// TIA Portal V19 export
FUNCTION "Input_Peripherie" : Void   // FC1010, LAD
TITLE = Input
{ S7_Optimized_Access := 'TRUE' }
// stored: AutoNumber false, SetENOAutomatically true
   VAR_TEMP
      Sperre_Inc_max : DInt;
      Sperre_Inc_min : DInt;
   END_VAR
BEGIN

REGION Network 1 (SCL): Schnelllauftor
   // Motorschutzschalter
   "Tor".In.MSS_ok := "E_MSS_ok_RT";
   // betriebsbereit
   "Tor".In.ok := "E_RT_ok";
   // Paneltasten
   "Tor".In.Knauf_Auto := "DB_ANLAGE".BA.Automat_ein;
   "Tor".In.T_auf := "Panel".RT.T_auf;
   "Tor".In.T_zu := "Panel".RT.T_zu;
   // Sensoren
   "Tor".In.S_auf := "E_S_RT_auf";
   "Tor".In.S_zu := "E_S_RT_zu";
   // --> Panel
   "Panel".RT.MSS_ok := "Tor".In.MSS_ok;
   "Panel".RT.ok := "Tor".In.ok;
   "Panel".RT.S_offen := "Tor".In.S_auf;
   "Panel".RT.S_geschlossen := "Tor".In.S_zu;
   // Automatik
   "Tor".In.Knauf_Auto := "DB_ANLAGE".BA.Automat_ein;
   // Fehlerquittung
   "Tor".In.ErrQ := "DB_ANLAGE".IN.Quitt_Err;
END_REGION

REGION Network 2 (SCL): Deckel
   REGION CM01
       // Sicherungen
       "Deckel_CM01".In.Si_24VDC_links := "E_Si_24VDC_CM01.MM01";
       "Deckel_CM01".In.Si_24VDC_rechts := "E_Si_24VDC_CM01.MM02";
       // Stellrückmeldungen
       "Deckel_CM01".In.SRM_links_auf := "E_Dkl_li_auf_CM01";
       "Deckel_CM01".In.SRM_links_zu := "E_Dkl_li_zu_CM01";
       "Deckel_CM01".In.SRM_rechts_auf := "E_Dkl_re_auf_CM01";
       "Deckel_CM01".In.SRM_rechts_zu := "E_Dkl_re_zu_CM01";
       // Sensoren
       "Deckel_CM01".In.S_links_auf := "E_S_Dkl_li_auf_CM01.BG01" AND NOT "E_S_Dkl_li_zu_CM01.BG02";
       "Deckel_CM01".In.S_links_zu := "E_S_Dkl_li_zu_CM01.BG02" AND NOT "E_S_Dkl_li_auf_CM01.BG01";
       "Deckel_CM01".In.S_rechts_auf := "E_S_Dkl_re_auf_CM01.BG03" AND NOT "E_S_Dkl_re_zu_CM01.BG04";
       "Deckel_CM01".In.S_rechts_zu := "E_S_Dkl_re_zu_CM01.BG04" AND NOT "E_S_Dkl_re_auf_CM01.BG03";
       // Bedienung via Panel
       "Deckel_CM01".In.Auto := "Panel".Deckel.CM01.Auto;
       "Deckel_CM01".In.Hand := "Panel".Deckel.CM01.Hand;
       "Deckel_CM01".In.Tipp := "Panel".Deckel.CM01.Tipp;

       "Deckel_CM01".In.T_links_auf := "Panel".Deckel.CM01.links_auf;
       "Deckel_CM01".In.T_links_zu := "Panel".Deckel.CM01.links_zu;
       "Deckel_CM01".In.T_rechts_auf := "Panel".Deckel.CM01.rechts_auf;
       "Deckel_CM01".In.T_rechts_zu := "Panel".Deckel.CM01.rechts_zu;
       // --> Panel
       "Panel".Deckel.CM01.SRM_links_auf := "Deckel_CM01".In.SRM_links_auf;
       "Panel".Deckel.CM01.SRM_links_zu := "Deckel_CM01".In.SRM_links_zu;
       "Panel".Deckel.CM01.SRM_rechts_auf := "Deckel_CM01".In.SRM_rechts_auf;
       "Panel".Deckel.CM01.SRM_rechts_zu := "Deckel_CM01".In.SRM_rechts_zu;
       "Panel".Deckel.CM01.S_links_auf := "Deckel_CM01".In.S_links_auf;
       "Panel".Deckel.CM01.S_links_zu := "Deckel_CM01".In.S_links_zu;
       "Panel".Deckel.CM01.S_rechts_auf := "Deckel_CM01".In.S_rechts_auf;
       "Panel".Deckel.CM01.S_rechts_zu := "Deckel_CM01".In.S_rechts_zu;
       "Panel".Deckel.CM01.Ist_Pos_links := "Deckel_CM01".Zst.Ist_Pos_links;
       "Panel".Deckel.CM01.Ist_Pos_rechts := "Deckel_CM01".Zst.Ist_Pos_rechts;

       // Transportwagen im sicheren Bereich
       IF "DB_Sperrbereiche".Sperre_links OR "DB_Sperrbereiche".Sperre_rechts THEN
           IF "DI_FW_1".OUT.VOR THEN
               "Deckel_CM01".Zst.TW_sicher := "DI_FW_1".ZST.PosInc >= ("DB_Sperrbereiche".Bereich[3].max_Inc + "DI_FW_1".PAR.Fahrt.Bereich_Pos);
           ELSE
               "Deckel_CM01".Zst.TW_sicher := "DI_FW_1".ZST.PosInc >= ("DB_Sperrbereiche".Bereich[3].max_Inc + "DI_FW_1".PAR.Fahrt.Bereich_lngsm);
           END_IF;
       ELSIF "DI_FW_1".OUT.VOR THEN
           "Deckel_CM01".Zst.TW_sicher := "DI_FW_1".ZST.PosInc >= ("DB_Sperrbereiche".Bereich[1].max_Inc + "DI_FW_1".PAR.Fahrt.Bereich_Pos);
       ELSE
           "Deckel_CM01".Zst.TW_sicher := "DI_FW_1".ZST.PosInc >= ("DB_Sperrbereiche".Bereich[1].max_Inc + "DI_FW_1".PAR.Fahrt.Bereich_lngsm);
       END_IF;

       // Fehlerquittung
       "Deckel_CM01".In.ErrQ := "DB_ANLAGE".IN.Quitt_Err;
   END_REGION ;
   REGION CM02
       // Sicherungen
       "Deckel_CM02".In.Si_24VDC_links := "E_Si_24VDC_CM02.MM03";
       "Deckel_CM02".In.Si_24VDC_rechts := "E_Si_24VDC_CM02.MM04";
       // Stellrückmeldungen
       "Deckel_CM02".In.SRM_links_auf := "E_Dkl_li_auf_CM02";
       "Deckel_CM02".In.SRM_links_zu := "E_Dkl_li_zu_CM02";
       "Deckel_CM02".In.SRM_rechts_auf := "E_Dkl_re_auf_CM02";
       "Deckel_CM02".In.SRM_rechts_zu := "E_Dkl_re_zu_CM02";
       // Sensoren
       "Deckel_CM02".In.S_links_auf := "E_S_Dkl_li_auf_CM02.BG12" AND NOT "E_S_Dkl_li_zu_CM02.BG13";
       "Deckel_CM02".In.S_links_zu := "E_S_Dkl_li_zu_CM02.BG13" AND NOT "E_S_Dkl_li_auf_CM02.BG12";
       "Deckel_CM02".In.S_rechts_auf := "E_S_Dkl_re_auf_CM02.BG14" AND NOT "E_S_Dkl_re_zu_CM02.BG15";
       "Deckel_CM02".In.S_rechts_zu := "E_S_Dkl_re_zu_CM02.BG15" AND NOT "E_S_Dkl_re_auf_CM02.BG14";
       // Bedienung via Panel
       "Deckel_CM02".In.Auto := "Panel".Deckel.CM02.Auto;
       "Deckel_CM02".In.Hand := "Panel".Deckel.CM02.Hand;
       "Deckel_CM02".In.Tipp := "Panel".Deckel.CM02.Tipp;

       "Deckel_CM02".In.T_links_auf := "Panel".Deckel.CM02.links_auf;
       "Deckel_CM02".In.T_links_zu := "Panel".Deckel.CM02.links_zu;
       "Deckel_CM02".In.T_rechts_auf := "Panel".Deckel.CM02.rechts_auf;
       "Deckel_CM02".In.T_rechts_zu := "Panel".Deckel.CM02.rechts_zu;
       // --> Panel
       "Panel".Deckel.CM02.SRM_links_auf := "Deckel_CM02".In.SRM_links_auf;
       "Panel".Deckel.CM02.SRM_links_zu := "Deckel_CM02".In.SRM_links_zu;
       "Panel".Deckel.CM02.SRM_rechts_auf := "Deckel_CM02".In.SRM_rechts_auf;
       "Panel".Deckel.CM02.SRM_rechts_zu := "Deckel_CM02".In.SRM_rechts_zu;
       "Panel".Deckel.CM02.S_links_auf := "Deckel_CM02".In.S_links_auf;
       "Panel".Deckel.CM02.S_links_zu := "Deckel_CM02".In.S_links_zu;
       "Panel".Deckel.CM02.S_rechts_auf := "Deckel_CM02".In.S_rechts_auf;
       "Panel".Deckel.CM02.S_rechts_zu := "Deckel_CM02".In.S_rechts_zu;
       "Panel".Deckel.CM02.Ist_Pos_links := "Deckel_CM02".Zst.Ist_Pos_links;
       "Panel".Deckel.CM02.Ist_Pos_rechts := "Deckel_CM02".Zst.Ist_Pos_rechts;

       // Transportwagen im sicheren Bereich
       IF "DB_Sperrbereiche".Sperre_links OR "DB_Sperrbereiche".Sperre_rechts THEN

           IF "DI_FW_1".OUT.VOR THEN
               "Deckel_CM02".Zst.TW_sicher :=
               ("DI_FW_1".ZST.PosInc <= ("DB_Sperrbereiche".Bereich[4].min_Inc - "DI_FW_1".PAR.Fahrt.Bereich_lngsm)) OR
               ("DI_FW_1".ZST.PosInc >= ("DB_Sperrbereiche".Bereich[4].max_Inc + "DI_FW_1".PAR.Fahrt.Bereich_Pos));

           ELSIF "DI_FW_1".OUT.RUECK THEN
               "Deckel_CM02".Zst.TW_sicher :=
               ("DI_FW_1".ZST.PosInc <= ("DB_Sperrbereiche".Bereich[4].min_Inc - "DI_FW_1".PAR.Fahrt.Bereich_Pos)) OR
               ("DI_FW_1".ZST.PosInc >= ("DB_Sperrbereiche".Bereich[4].max_Inc + "DI_FW_1".PAR.Fahrt.Bereich_lngsm));
           ELSE
               "Deckel_CM02".Zst.TW_sicher :=
               ("DI_FW_1".ZST.PosInc <= ("DB_Sperrbereiche".Bereich[4].min_Inc)) OR
               ("DI_FW_1".ZST.PosInc >= ("DB_Sperrbereiche".Bereich[4].max_Inc));
           END_IF;

       ELSIF "DI_FW_1".OUT.VOR THEN
           "Deckel_CM02".Zst.TW_sicher :=
           ("DI_FW_1".ZST.PosInc <= ("DB_Sperrbereiche".Bereich[2].min_Inc - "DI_FW_1".PAR.Fahrt.Bereich_lngsm)) OR
           ("DI_FW_1".ZST.PosInc >= ("DB_Sperrbereiche".Bereich[2].max_Inc + "DI_FW_1".PAR.Fahrt.Bereich_Pos));

       ELSIF "DI_FW_1".OUT.RUECK THEN
           "Deckel_CM02".Zst.TW_sicher :=
           ("DI_FW_1".ZST.PosInc <= ("DB_Sperrbereiche".Bereich[2].min_Inc - "DI_FW_1".PAR.Fahrt.Bereich_Pos)) OR
           ("DI_FW_1".ZST.PosInc >= ("DB_Sperrbereiche".Bereich[2].max_Inc + "DI_FW_1".PAR.Fahrt.Bereich_lngsm));

       ELSE
           "Deckel_CM02".Zst.TW_sicher :=
           ("DI_FW_1".ZST.PosInc <= ("DB_Sperrbereiche".Bereich[2].min_Inc)) OR
           ("DI_FW_1".ZST.PosInc >= ("DB_Sperrbereiche".Bereich[2].max_Inc));
       END_IF;

       // Fehlerquittung
       "Deckel_CM02".In.ErrQ := "DB_ANLAGE".IN.Quitt_Err;
   END_REGION ;
END_REGION

REGION Network 3 (SCL): CM01
   REGION Filtern
       "FP_CM01.GP01".Param.Name_Pumpe := 'FP_CM01.GP01';
       "FP_CM01.GP01".Param.Name_Filter := 'Filter HQ1';
       // Niveaus
       "FP_CM01.GP01".In.Niv_TLS := "E_Niv_TLS_CM01.BL04";
       "FP_CM01.GP01".In.Niv_min := "E_Niv_Min_CM01.BL03";
       "FP_CM01.GP01".In.Niv_max := "E_Niv_Max_CM01.BL02";
       "FP_CM01.GP01".In.Niv_Uel := NOT "E_Niv_UeL_CM01.BL01";
       "FP_CM01.GP01".In.Frg_Niv_CM05 := NOT "Pu_CM05.GP11_DB".In."Niv_max_CM05.BL01" AND NOT "Pu_CM05.GP11_DB".In."Niv_Uel_CM05.BL05";
       "FP_CM01.GP01".In.Leckage_ok := "E_LS_HQ0x.BL12";
       "FP_CM01.GP01".In.ext_Freigabe := "E_Al_Gas_ok" AND NOT "E_Not-Strom";
       // Ist-Druck Pumpe
       "FP_CM01.GP01".In.Druck_Pumpe := "Panel".IW."p_CM01.BP03";
       // Differenz-Druck Filter
       "FP_CM01.GP01".In.Delta_p_Filter := "Panel".IW."p_HQ01.BP01";

       //Stellrückmeldungen (Filtern)
       "FP_CM01.GP01".In.SRM_Saugseite_auf := "E_SRM_CM01.QM18_auf" AND NOT "E_SRM_CM01.QM18_zu";
       "FP_CM01.GP01".In.SRM_Saugseite_zu := "E_SRM_CM01.QM18_zu" AND NOT "E_SRM_CM01.QM18_auf";
       "FP_CM01.GP01".In.SRM_Eingang_Filter_auf := "E_SRM_HQ01.QM21_auf" AND NOT "E_SRM_HQ01.QM21_zu";
       "FP_CM01.GP01".In.SRM_Eingang_Filter_zu := "E_SRM_HQ01.QM21_zu" AND NOT "E_SRM_HQ01.QM21_auf";
       "FP_CM01.GP01".In.SRM_Ausgang_Filter_auf := "E_SRM_HQ01.QM23_auf" AND NOT "E_SRM_HQ01.QM23_zu";
       "FP_CM01.GP01".In.SRM_Ausgang_Filter_zu := "E_SRM_HQ01.QM23_zu" AND NOT "E_SRM_HQ01.QM23_auf";

       "FP_CM01.GP01".In.SRM_Eingang_Spülltg_P_auf := "E_SRM_CM01.QM19_auf" AND NOT "E_SRM_CM01.QM19_zu";
       "FP_CM01.GP01".In.SRM_Eingang_Spülltg_P_zu := "E_SRM_CM01.QM19_zu" AND NOT "E_SRM_CM01.QM19_auf";
       "FP_CM01.GP01".In.SRM_Eingang_Spülltg_F_auf := "E_SRM_HQ01.QM22_auf" AND NOT "E_SRM_HQ01.QM22_zu";
       "FP_CM01.GP01".In.SRM_Eingang_Spülltg_F_zu := "E_SRM_HQ01.QM22_zu" AND NOT "E_SRM_HQ01.QM22_auf";
       "FP_CM01.GP01".In.SRM_Ausgang_Spülltg_auf := "E_SRM_HQ01.QM24_auf" AND NOT "E_SRM_HQ01.QM24_zu";
       "FP_CM01.GP01".In.SRM_Ausgang_Spülltg_zu := "E_SRM_HQ01.QM24_zu" AND NOT "E_SRM_HQ01.QM24_auf";
       "FP_CM01.GP01".In.SRM_Entluften_auf := "E_SRM_HQ01.LV01_auf" AND NOT "E_SRM_HQ01.LV01_zu";
       "FP_CM01.GP01".In.SRM_Entlueften_zu := "E_SRM_HQ01.LV01_zu" AND NOT "E_SRM_HQ01.LV01_auf";

       // Filtergehäuse
       "FP_CM01.GP01".In.GW_p_FG := "E_GW_p_HQ01.BP01";
       "FP_CM01.GP01".In.Sensor_FG_links := "E_S_FG_li_HQ01.BG07";
       "FP_CM01.GP01".In.Sensor_FG_rechts := "E_S_FG_re_HQ01.BG08";
       "FP_CM01.GP01".In.Einhausung_HQ0x_zu := "DB_PNOZ_IN_Out".In.FG_zu_HQ01;
       "FP_CM01.GP01".Param.WarnGr_FW := "Panel".HQ01.WarnGr_FW;
       "FP_CM01.GP01".Param.Wechsel_FW := "Panel".HQ01.Wechsel_FW;

       // Not-Halt
       "FP_CM01.GP01".In.NotHalt := NOT "DB_PNOZ_IN_Out".In.NH_Frg_FP_CM01;

       "FP_CM01.GP01".In.GW_p_FP := "E_GW_p_CM01.BP03";
       "FP_CM01.GP01".In.GW_LF_FP := "E_GW_LF_CM01.BN01";

       // Frequenzumrichter [Index 1] 
       "FP_CM01.GP01".In.FU_speed := "FU_In_Out".FU[1].PE.Speed;
       "FP_CM01.GP01".In.FU_betriebsbereit := "FU_In_Out".FU[1].PE.Statusbyte.Bereit;
       "FP_CM01.GP01".In.FU_Stoerung := "FU_In_Out".FU[1].PE.Statusbyte.Stoer;
       "FP_CM01.GP01".Param.SW_Hand := "Panel".FP_CM01.SW_Hand;
       "FP_CM01.GP01".Param.SW_Auto_AZ := "Panel".FP_CM01.SW_Auto_AZ;
       "FP_CM01.GP01".Param.SW_Auto_aAZ := "Panel".FP_CM01.SW_Auto_aAZ;

       // Hand
       "FP_CM01.GP01".In.Ein := "Panel".FP_CM01.Ein;
       // Auto
       "FP_CM01.GP01".In.Auto := "Panel".FP_CM01.Auto;
       // Betriebsart
       "FP_CM01.GP01".In.Betriebsart := "Panel".FP_CM01.BA;
       // Spülzeit
       "FP_CM01.GP01".Param.Spülzeit_Pumpe := DINT_TO_TIME(INT_TO_DINT("Panel".FP_CM01.Sp_Ventil.Sollzeit) * 1000);
       // Zeiten Filterwechsel
       "FP_CM01.GP01".Param.FG_Zeit_leeren_Saurebecken := DINT_TO_TIME(INT_TO_DINT("Panel".FP_CM01.Sp_Filter.Zeit_leeren_Saure) * 1000);
       "FP_CM01.GP01".Param.FG_Zeit_leeren_CM05 := DINT_TO_TIME(INT_TO_DINT("Panel".FP_CM01.Sp_Filter.Zeit_leeren_CM05) * 1000);
       "FP_CM01.GP01".Param.FW_Spülzeit := DINT_TO_TIME(INT_TO_DINT("Panel".FP_CM01.Sp_Filter.Zeit_Spülen) * 1000);
       "FP_CM01.GP01".Param.FW_Wartezeit := DINT_TO_TIME(INT_TO_DINT("Panel".FP_CM01.Sp_Filter.Wartezeit) * 1000);
       "FP_CM01.GP01".Param.FW_Zeit_fuellen := DINT_TO_TIME(INT_TO_DINT("Panel".FP_CM01.Sp_Filter.Zeit_füllen) * 1000);
       // Drucktest Pumpe
       "FP_CM01.GP01".Param.DT_Druckaufbau := T#1m;
       "FP_CM01.GP01".Param.SW_Drucktest_Pumpe := "Panel".FP_CM01.Drucktest_Pumpe.Solldruck;
       "FP_CM01.GP01".Param.DT_Testzeit_Pumpe := DINT_TO_TIME(INT_TO_DINT("Panel".FP_CM01.Drucktest_Pumpe.Sollzeit) * 1000);
       // Drucktest Filter
       "FP_CM01.GP01".Param.DT_Druckaufbau := T#1m;
       "FP_CM01.GP01".Param.SW_Drucktest_Filter := "Panel".FP_CM01.Drucktest_Filter.Solldruck;
       "FP_CM01.GP01".Param.DT_Testzeit_Filter := DINT_TO_TIME(INT_TO_DINT("Panel".FP_CM01.Drucktest_Filter.Sollzeit) * 1000);

       IF "Panel".HQ01.Quitt_FW THEN
           "FP_CM01.GP01".In.Quitt_FW := TRUE;
           "Panel".HQ01.Quitt_FW := FALSE;
       END_IF;

       //--> Panel
       "Panel".CM01.GW_p_FP := "FP_CM01.GP01".Mld.GW_p_FP;
       "Panel".CM01.GW_LF_FP := "FP_CM01.GP01".Mld.GW_LF_FP;

       "Panel".FP_CM01.Sp_Ventil.Restzeit := TIME_TO_INT("FP_CM01.GP01".Zst.Restzeit_Spülen_Pumpe / 1000);
       "Panel".FP_CM01.Sp_Filter.Restzeit := TIME_TO_INT("FP_CM01.GP01".Zst.Restzeit_Filter / 1000);
       "Panel".FP_CM01.Drucktest_Pumpe.Restzeit := TIME_TO_INT("FP_CM01.GP01".Zst.Restzeit_DT / 1000);
       "Panel".FP_CM01.Drucktest_Pumpe.Schritt := "FP_CM01.GP01".Zst.Status_DT_Pumpe;
       "Panel".FP_CM01.Status_FW := "FP_CM01.GP01".Zst.Status_FW;

       "Panel".FP_CM01.Bedienung_Erlaubt := "FP_CM01.GP01".Zst.Bedienung_erlaubt;

       "Panel".FP_CM01.Status := "FP_CM01.GP01".Zst.Status_GP0x;
       "Panel".FP_CM01.speed := "FP_CM01.GP01".Zst.speed;

       "Panel".HQ01.S_Dkl_FG_li := "FP_CM01.GP01".In.Sensor_FG_links;
       "Panel".HQ01.S_Dkl_FG_re := "FP_CM01.GP01".In.Sensor_FG_rechts;
       "Panel".HQ01.S_FG_zu := "FP_CM01.GP01".In.Einhausung_HQ0x_zu;
       "Panel".HQ01.Niv_Leckage := NOT "FP_CM01.GP01".In.Leckage_ok;
       "Panel".HQ01.Quitt_FW_erlaubt := "FP_CM01.GP01".In.Sensor_FG_links AND "FP_CM01.GP01".In.Sensor_FG_rechts AND
       "FP_CM01.GP01".In.Einhausung_HQ0x_zu AND "FP_CM01.GP01".Mld.FG_Spülen_Ende AND "FP_CM01.GP01".Zst.Status_FW = 5;

       "Panel".FP_CM01.Drucktest_Filter.Restzeit := TIME_TO_INT("FP_CM01.GP01".Zst.Restzeit_DT / 1000);
       "Panel".FP_CM01.Drucktest_Filter.Schritt := "FP_CM01.GP01".Zst.Status_DT_Filter;
   END_REGION

   REGION Umwälzen
       "UP_CM01.GP02".Param.Name := 'UP_CM01.GP02';
       // Niveaus
       "UP_CM01.GP02".In.Niv_TLS := "E_Niv_TLS_CM01.BL04";
       "UP_CM01.GP02".In.Niv_min := "E_Niv_Min_CM01.BL03";
       "UP_CM01.GP02".In.Niv_max := "E_Niv_Max_CM01.BL02";
       "UP_CM01.GP02".In.Niv_Uel := NOT "E_Niv_UeL_CM01.BL01";
       "UP_CM01.GP02".In.Frg_Niv_CM05 := NOT "Pu_CM05.GP11_DB".In."Niv_max_CM05.BL01" AND NOT "Pu_CM05.GP11_DB".In."Niv_Uel_CM05.BL05";
       "UP_CM01.GP02".In.ext_Freigabe := "E_Al_Gas_ok" AND NOT "E_Not-Strom";
       // Ist-Druck
       "UP_CM01.GP02".In.Druck_Pumpe := "Panel".IW."p_CM01.BP04";

       //Stellrückmeldungen (Umwälzen)
       "UP_CM01.GP02".In.SRM_Saugseite_auf := "E_SRM_CM01.QM25_auf" AND NOT "E_SRM_CM01.QM25_zu";
       "UP_CM01.GP02".In.SRM_Saugseite_zu := "E_SRM_CM01.QM25_zu" AND NOT "E_SRM_CM01.QM25_auf";
       "UP_CM01.GP02".In.SRM_Druckseite_auf := "E_SRM_CM01.QM26_auf" AND NOT "E_SRM_CM01.QM26_zu";
       "UP_CM01.GP02".In.SRM_Druckseite_zu := "E_SRM_CM01.QM26_zu" AND NOT "E_SRM_CM01.QM26_auf";
       "UP_CM01.GP02".In.SRM_Eingang_Spülltg_auf := "E_SRM_CM01.QM20_auf" AND NOT "E_SRM_CM01.QM20_zu";
       "UP_CM01.GP02".In.SRM_Eingang_Spülltg_zu := "E_SRM_CM01.QM20_zu" AND NOT "E_SRM_CM01.QM20_auf";
       "UP_CM01.GP02".In.SRM_Ausgang_Spülltg_auf := "E_SRM_CM01.QM27_auf" AND NOT "E_SRM_CM01.QM27_zu";
       "UP_CM01.GP02".In.SRM_Ausgang_Spülltg_zu := "E_SRM_CM01.QM27_zu" AND NOT "E_SRM_CM01.QM27_auf";
       "UP_CM01.GP02".In.SRM_Entsogung_UV02_auf := "E_SRM_GP02.QM45_auf" AND NOT "E_SRM_GP02.QM45_zu";
       "UP_CM01.GP02".In.SRM_Entsogung_UV02_zu := "E_SRM_GP02.QM45_zu" AND NOT "E_SRM_GP02.QM45_auf";
       "UP_CM01.GP02".In.SRM_UV02_GP01_auf := "DB_PNOZ_IN_Out".In."SRM_Auf_BG-QM44" AND NOT "DB_PNOZ_IN_Out".In."SRM_Zu_BG-QM44";
       "UP_CM01.GP02".In.SRM_UV02_GP01_zu := "DB_PNOZ_IN_Out".In."SRM_Zu_BG-QM44" AND NOT "DB_PNOZ_IN_Out".In."SRM_Auf_BG-QM44";
       "UP_CM01.GP02".In.SRM_UV02_GP02_auf := "DB_PNOZ_IN_Out".In."SRM_Auf_BG-QM43" AND NOT "DB_PNOZ_IN_Out".In."SRM_Zu_BG-QM43";
       "UP_CM01.GP02".In.SRM_UV02_GP02_zu := "DB_PNOZ_IN_Out".In."SRM_Zu_BG-QM43" AND NOT "DB_PNOZ_IN_Out".In."SRM_Auf_BG-QM43";
       "UP_CM01.GP02".In."SRM_GP02.QM41_auf" := "E_SRM_GP02.QM41_auf" AND NOT "E_SRM_GP02.QM41_zu";
       "UP_CM01.GP02".In."SRM_GP01.QM14_auf" := "E_SRM_GP01.QM14_auf" AND NOT "E_SRM_GP01.QM14_zu";

       // Türen GP0x
       "UP_CM01.GP02".In.Tuer_zu_Seite_GP01 := "DB_PNOZ_IN_Out".In.Tuer_zu_Seite_GP01;
       "UP_CM01.GP02".In.Tuer_zu_vorn_GP01 := "DB_PNOZ_IN_Out".In.Tuer_zu_vorn_GP01;
       "UP_CM01.GP02".In.Tuer_zu_vorn_GP02 := "DB_PNOZ_IN_Out".In.Tuer_zu_vorn_GP02;
       // Leckagen Entsorgung
       "UP_CM01.GP02".In.Leckage_Doppelrohr_ok_BL26 := "E_LS_GP02.BL26";
       "UP_CM01.GP02".In.Leckage_Doppelschlauch_ok_BL33 := "E_LS_GP02.BL33";
       "UP_CM01.GP02".In.Leckage_Uml_Tunnel_ok_BL34 := "E_LS_GP01.BL34";
       "UP_CM01.GP02".In.Leckage_PFA_Uebergang_ok_BL16 := "E_LS_GP01.BL16";
       "UP_CM01.GP02".In.Leckage_PFA_Uebergang_ok_BL25 := "E_LS_GP02.BL25";

       "UP_CM01.GP02".In.Imp_Dfl := "E_Imp_GP02.BF02";
       "UP_CM01.GP02".In.Quitt_Al_Dfl := "DB_ANLAGE".IN.Quitt_Err;

       "UP_CM01.GP02".In.GW_p_UP := "E_GW_p_CM01.BP04";
       "UP_CM01.GP02".In.GW_LF_UP := "E_GW_LF_CM01.BN02";
       "UP_CM01.GP02".In.GW_Dfl := "E_GW_Dfl_GP02.BF02";
       // TW senkt
       "UP_CM01.GP02".In.TW_senkt := ("DB_POS".POS[1].FW_Senkt OR "DB_POS".POS[2].FW_Senkt OR "DB_POS".POS[3].FW_Senkt
       OR "DB_POS".POS[4].FW_Senkt OR "DB_POS".POS[5].FW_Senkt OR "DB_POS".POS[6].FW_Senkt) AND "DI_FW_1".ZST.Mittig;

       // Frequenzumrichter [Index 2] Umwälzen
       "UP_CM01.GP02".In.FU_speed := "FU_In_Out".FU[2].PE.Speed;
       "UP_CM01.GP02".In.FU_betriebsbereit := "FU_In_Out".FU[2].PE.Statusbyte.Bereit;
       "UP_CM01.GP02".In.FU_Stoerung := "FU_In_Out".FU[2].PE.Statusbyte.Stoer;
       "UP_CM01.GP02".Param.SW_Hand := "Panel".UP_CM01.SW_Hand;
       "UP_CM01.GP02".Param.SW_Auto_AZ := "Panel".UP_CM01.SW_Auto_AZ;
       "UP_CM01.GP02".Param.SW_Auto_aAZ := "Panel".UP_CM01.SW_Auto_aAZ;

       // Hand
       "UP_CM01.GP02".In.Ein := "Panel".UP_CM01.Ein;
       // Auto
       "UP_CM01.GP02".In.Auto := "Panel".UP_CM01.Auto;
       // Betriebsart
       "UP_CM01.GP02".In.Betriebsart := "Panel".UP_CM01.BA;
       // Spülzeit
       "UP_CM01.GP02".Param.Spülzeit := DINT_TO_TIME(INT_TO_DINT("Panel".UP_CM01.Sp_Ventil.Sollzeit) * 1000);
       // Drucktest
       "UP_CM01.GP02".Param.DT_Druckaufbau := T#1m;
       "UP_CM01.GP02".Param.SW_Drucktest := "Panel".UP_CM01.Drucktest.Solldruck;
       "UP_CM01.GP02".Param.DT_Testzeit := DINT_TO_TIME(INT_TO_DINT("Panel".UP_CM01.Drucktest.Sollzeit) * 1000);

       //--> Panel
       "Panel".CM01.Niv_TGS := "UP_CM01.GP02".In.Niv_TLS;
       "Panel".CM01.Niv_Min := "UP_CM01.GP02".In.Niv_min;
       "Panel".CM01.Niv_max := "UP_CM01.GP02".In.Niv_max;
       "Panel".CM01.Niv_Uel := "UP_CM01.GP02".Mld.Niv_Ueberlauf;
       "Panel".CM01.GW_p_UP := "UP_CM01.GP02".Mld.GW_p_UP;
       "Panel".CM01.GW_LF_UP := "UP_CM01.GP02".Mld.GW_LF_UP;
       "Panel".CM01.Niv_Proz := "UP_CM01.GP02".Zst.Niveau;
       "Panel".UP_CM01.Sp_Ventil.Restzeit := TIME_TO_INT("UP_CM01.GP02".Zst.Restzeit_Spülen / 1000);
       "Panel".UP_CM01.Drucktest.Restzeit := TIME_TO_INT("UP_CM01.GP02".Zst.Restzeit_DT / 1000);
       "Panel".UP_CM01.Drucktest.Schritt := "UP_CM01.GP02".Zst.Status_DT;
       "Panel".UP_CM01.Status := "UP_CM01.GP02".Zst.Status_GP0x;
       "Panel".UP_CM01.speed := "UP_CM01.GP02".Zst.speed;
       "Panel".UP_CM01.Bedienung_Erlaubt := "UP_CM01.GP02".Zst.Bedienung_erlaubt;
   END_REGION
END_REGION

REGION Network 4 (SCL): CM02
   REGION Filtern
       "FP_CM02.GP04".Param.Name_Pumpe := 'FP_CM02.GP04';
       "FP_CM02.GP04".Param.Name_Filter := 'Filter HQ2';
       // Niveaus
       "FP_CM02.GP04".In.Niv_TLS := "E_Niv_TLS_CM02.BL11";
       "FP_CM02.GP04".In.Niv_min := "E_Niv_Min_CM02.BL10";
       "FP_CM02.GP04".In.Niv_max := "E_Niv_Max_CM02.BL09";
       "FP_CM02.GP04".In.Niv_Uel := NOT "E_Niv_UeL_CM02.BL08";
       "FP_CM02.GP04".In.Frg_Niv_CM05 := NOT "Pu_CM05.GP11_DB".In."Niv_max_CM05.BL01" AND NOT "Pu_CM05.GP11_DB".In."Niv_Uel_CM05.BL05";
       "FP_CM02.GP04".In.Leckage_ok := "E_LS_HQ0x.BL12";
       "FP_CM02.GP04".In.ext_Freigabe := "E_Al_Gas_ok" AND NOT "E_Not-Strom";
       // Ist-Druck Pumpe
       "FP_CM02.GP04".In.Druck_Pumpe := "Panel".IW."p_CM02.BP06";
       // Differenz-Druck Filter
       "FP_CM02.GP04".In.Delta_p_Filter := "Panel".IW."p_HQ02.BP02";

       //Stellrückmeldungen (Filtern)
       "FP_CM02.GP04".In.SRM_Saugseite_auf := "E_SRM_CM02.QM55_auf" AND NOT "E_SRM_CM02.QM55_zu";
       "FP_CM02.GP04".In.SRM_Saugseite_zu := "E_SRM_CM02.QM55_zu" AND NOT "E_SRM_CM02.QM55_auf";
       "FP_CM02.GP04".In.SRM_Eingang_Filter_auf := "E_SRM_HQ02.QM59_auf" AND NOT "E_SRM_HQ02.QM59_zu";
       "FP_CM02.GP04".In.SRM_Eingang_Filter_zu := "E_SRM_HQ02.QM59_zu" AND NOT "E_SRM_HQ02.QM59_auf";
       "FP_CM02.GP04".In.SRM_Ausgang_Filter_auf := "E_SRM_HQ02.QM60_auf" AND NOT "E_SRM_HQ02.QM60_zu";
       "FP_CM02.GP04".In.SRM_Ausgang_Filter_zu := "E_SRM_HQ02.QM60_zu" AND NOT "E_SRM_HQ02.QM60_auf";

       "FP_CM02.GP04".In.SRM_Eingang_Spülltg_P_auf := "E_SRM_CM02.QM56_auf" AND NOT "E_SRM_CM02.QM56_zu";
       "FP_CM02.GP04".In.SRM_Eingang_Spülltg_P_zu := "E_SRM_CM02.QM56_zu" AND NOT "E_SRM_CM02.QM56_auf";
       "FP_CM02.GP04".In.SRM_Eingang_Spülltg_F_auf := "E_SRM_HQ02.QM58_auf" AND NOT "E_SRM_HQ02.QM58_zu";
       "FP_CM02.GP04".In.SRM_Eingang_Spülltg_F_zu := "E_SRM_HQ02.QM58_zu" AND NOT "E_SRM_HQ02.QM58_auf";
       "FP_CM02.GP04".In.SRM_Ausgang_Spülltg_auf := "E_SRM_HQ02.QM61_auf" AND NOT "E_SRM_HQ02.QM61_zu";
       "FP_CM02.GP04".In.SRM_Ausgang_Spülltg_zu := "E_SRM_HQ02.QM61_zu" AND NOT "E_SRM_HQ02.QM61_auf";
       "FP_CM02.GP04".In.SRM_Entluften_auf := "E_SRM_HQ02.LV02_auf" AND NOT "E_SRM_HQ02.LV02_zu";
       "FP_CM02.GP04".In.SRM_Entlueften_zu := "E_SRM_HQ02.LV02_zu" AND NOT "E_SRM_HQ02.LV02_auf";

       // Filtergehäuse
       "FP_CM02.GP04".In.GW_p_FG := "E_GW_p_HQ02.BP02";
       "FP_CM02.GP04".In.Sensor_FG_links := "E_S_FG_li_HQ02.BG10";
       "FP_CM02.GP04".In.Sensor_FG_rechts := "E_S_FG_re_HQ02.BG11";
       "FP_CM02.GP04".In.Einhausung_HQ0x_zu := "DB_PNOZ_IN_Out".In.FG_zu_HQ02;
       "FP_CM02.GP04".Param.WarnGr_FW := "Panel".HQ02.WarnGr_FW;
       "FP_CM02.GP04".Param.Wechsel_FW := "Panel".HQ02.Wechsel_FW;

       // Not-Halt
       "FP_CM02.GP04".In.NotHalt := NOT "DB_PNOZ_IN_Out".In.NH_Frg_FP_CM02;

       "FP_CM02.GP04".In.GW_p_FP := "E_GW_p_CM02.BP06";
       "FP_CM02.GP04".In.GW_LF_FP := "E_GW_LF_CM02.BN03";

       // Frequenzumrichter [Index 4] 
       "FP_CM02.GP04".In.FU_speed := "FU_In_Out".FU[4].PE.Speed;
       "FP_CM02.GP04".In.FU_betriebsbereit := "FU_In_Out".FU[4].PE.Statusbyte.Bereit;
       "FP_CM02.GP04".In.FU_Stoerung := "FU_In_Out".FU[4].PE.Statusbyte.Stoer;
       "FP_CM02.GP04".Param.SW_Hand := "Panel".FP_CM02.SW_Hand;
       "FP_CM02.GP04".Param.SW_Auto_AZ := "Panel".FP_CM02.SW_Auto_AZ;
       "FP_CM02.GP04".Param.SW_Auto_aAZ := "Panel".FP_CM02.SW_Auto_aAZ;

       // Hand
       "FP_CM02.GP04".In.Ein := "Panel".FP_CM02.Ein;
       // Auto
       "FP_CM02.GP04".In.Auto := "Panel".FP_CM02.Auto;
       // Betriebsart
       "FP_CM02.GP04".In.Betriebsart := "Panel".FP_CM02.BA;
       // Spülzeit
       "FP_CM02.GP04".Param.Spülzeit_Pumpe := DINT_TO_TIME(INT_TO_DINT("Panel".FP_CM02.Sp_Ventil.Sollzeit) * 1000);
       // Zeiten Filterwechsel
       "FP_CM02.GP04".Param.FG_Zeit_leeren_Saurebecken := DINT_TO_TIME(INT_TO_DINT("Panel".FP_CM02.Sp_Filter.Zeit_leeren_Saure) * 1000);
       "FP_CM02.GP04".Param.FG_Zeit_leeren_CM05 := DINT_TO_TIME(INT_TO_DINT("Panel".FP_CM02.Sp_Filter.Zeit_leeren_CM05) * 1000);
       "FP_CM02.GP04".Param.FW_Spülzeit := DINT_TO_TIME(INT_TO_DINT("Panel".FP_CM02.Sp_Filter.Zeit_Spülen) * 1000);
       "FP_CM02.GP04".Param.FW_Wartezeit := DINT_TO_TIME(INT_TO_DINT("Panel".FP_CM02.Sp_Filter.Wartezeit) * 1000);
       "FP_CM02.GP04".Param.FW_Zeit_fuellen := DINT_TO_TIME(INT_TO_DINT("Panel".FP_CM02.Sp_Filter.Zeit_füllen) * 1000);
       "Panel".FP_CM02.Status_FW := "FP_CM02.GP04".Zst.Status_FW;
       // Drucktest Pumpe
       "FP_CM02.GP04".Param.DT_Druckaufbau := T#1m;
       "FP_CM02.GP04".Param.SW_Drucktest_Pumpe := "Panel".FP_CM02.Drucktest_Pumpe.Solldruck;
       "FP_CM02.GP04".Param.DT_Testzeit_Pumpe := DINT_TO_TIME(INT_TO_DINT("Panel".FP_CM02.Drucktest_Pumpe.Sollzeit) * 1000);
       // Drucktest Filter
       "FP_CM02.GP04".Param.DT_Druckaufbau := T#1m;
       "FP_CM02.GP04".Param.SW_Drucktest_Filter := "Panel".FP_CM02.Drucktest_Filter.Solldruck;
       "FP_CM02.GP04".Param.DT_Testzeit_Filter := DINT_TO_TIME(INT_TO_DINT("Panel".FP_CM02.Drucktest_Filter.Sollzeit) * 1000);

       IF "Panel".HQ02.Quitt_FW THEN
           "FP_CM02.GP04".In.Quitt_FW := TRUE;
           "Panel".HQ02.Quitt_FW := FALSE;
       END_IF;

       //--> Panel
       "Panel".CM02.GW_p_FP := "FP_CM02.GP04".Mld.GW_p_FP;
       "Panel".CM02.GW_LF_FP := "FP_CM02.GP04".Mld.GW_LF_FP;

       "Panel".FP_CM02.Sp_Ventil.Restzeit := TIME_TO_INT("FP_CM02.GP04".Zst.Restzeit_Spülen_Pumpe / 1000);
       "Panel".FP_CM02.Sp_Filter.Restzeit := TIME_TO_INT("FP_CM02.GP04".Zst.Restzeit_Filter / 1000);
       "Panel".FP_CM02.Drucktest_Pumpe.Restzeit := TIME_TO_INT("FP_CM02.GP04".Zst.Restzeit_DT / 1000);
       "Panel".FP_CM02.Drucktest_Pumpe.Schritt := "FP_CM02.GP04".Zst.Status_DT_Pumpe;
       "Panel".FP_CM02.Status := "FP_CM02.GP04".Zst.Status_GP0x;
       "Panel".FP_CM02.speed := "FP_CM02.GP04".Zst.speed;

       "Panel".FP_CM02.Bedienung_Erlaubt := "FP_CM02.GP04".Zst.Bedienung_erlaubt;

       "Panel".HQ02.S_Dkl_FG_li := "FP_CM02.GP04".In.Sensor_FG_links;
       "Panel".HQ02.S_Dkl_FG_re := "FP_CM02.GP04".In.Sensor_FG_rechts;
       "Panel".HQ02.S_FG_zu := "FP_CM02.GP04".In.Einhausung_HQ0x_zu;
       "Panel".HQ02.Niv_Leckage := NOT "FP_CM02.GP04".In.Leckage_ok;

       "Panel".HQ02.Quitt_FW_erlaubt := "FP_CM02.GP04".In.Sensor_FG_links AND "FP_CM02.GP04".In.Sensor_FG_rechts AND
       "FP_CM02.GP04".In.Einhausung_HQ0x_zu AND "FP_CM02.GP04".Mld.FG_Spülen_Ende AND "FP_CM02.GP04".Zst.Status_FW = 5;

       "Panel".FP_CM02.Drucktest_Filter.Restzeit := TIME_TO_INT("FP_CM02.GP04".Zst.Restzeit_DT / 1000);
       "Panel".FP_CM02.Drucktest_Filter.Schritt := "FP_CM02.GP04".Zst.Status_DT_Filter;
   END_REGION

   REGION Umwälzen
       "UP_CM02.GP05".Param.Name := 'UP_CM02.GP05';
       // Niveaus
       "UP_CM02.GP05".In.Niv_TLS := "E_Niv_TLS_CM02.BL11";
       "UP_CM02.GP05".In.Niv_min := "E_Niv_Min_CM02.BL10";
       "UP_CM02.GP05".In.Niv_max := "E_Niv_Max_CM02.BL09";
       "UP_CM02.GP05".In.Niv_Uel := NOT "E_Niv_UeL_CM02.BL08";
       "UP_CM02.GP05".In.Frg_Niv_CM05 := NOT "Pu_CM05.GP11_DB".In."Niv_max_CM05.BL01" AND NOT "Pu_CM05.GP11_DB".In."Niv_Uel_CM05.BL05";
       "UP_CM02.GP05".In.ext_Freigabe := "E_Al_Gas_ok" AND NOT "E_Not-Strom";
       // Ist-Druck
       "UP_CM02.GP05".In.Druck_Pumpe := "Panel".IW."p_CM02.BP07";

       //Stellrückmeldungen
       "UP_CM02.GP05".In.SRM_Saugseite_auf := "E_SRM_CM02.QM62_auf" AND NOT "E_SRM_CM02.QM62_zu";
       "UP_CM02.GP05".In.SRM_Saugseite_zu := "E_SRM_CM02.QM62_zu" AND NOT "E_SRM_CM02.QM62_auf";
       "UP_CM02.GP05".In.SRM_Druckseite_auf := "E_SRM_CM02.QM63_auf" AND NOT "E_SRM_CM02.QM63_zu";
       "UP_CM02.GP05".In.SRM_Druckseite_zu := "E_SRM_CM02.QM63_zu" AND NOT "E_SRM_CM02.QM63_auf";
       "UP_CM02.GP05".In.SRM_Eingang_Spülltg_auf := "E_SRM_CM02.QM57_auf" AND NOT "E_SRM_CM02.QM57_zu";
       "UP_CM02.GP05".In.SRM_Eingang_Spülltg_zu := "E_SRM_CM02.QM57_zu" AND NOT "E_SRM_CM02.QM57_auf";
       "UP_CM02.GP05".In.SRM_Ausgang_Spülltg_auf := "E_SRM_CM02.QM64_auf" AND NOT "E_SRM_CM02.QM64_zu";
       "UP_CM02.GP05".In.SRM_Ausgang_Spülltg_zu := "E_SRM_CM02.QM64_zu" AND NOT "E_SRM_CM02.QM64_auf";
       "UP_CM02.GP05".In.SRM_Entsogung_UV02_auf := "E_SRM_GP02.QM46_auf" AND NOT "E_SRM_GP02.QM46_zu";
       "UP_CM02.GP05".In.SRM_Entsogung_UV02_zu := "E_SRM_GP02.QM46_zu" AND NOT "E_SRM_GP02.QM46_auf";
       "UP_CM02.GP05".In.SRM_UV02_GP01_auf := "DB_PNOZ_IN_Out".In."SRM_Auf_BG-QM44" AND NOT "DB_PNOZ_IN_Out".In."SRM_Zu_BG-QM44";
       "UP_CM02.GP05".In.SRM_UV02_GP01_zu := "DB_PNOZ_IN_Out".In."SRM_Zu_BG-QM44" AND NOT "DB_PNOZ_IN_Out".In."SRM_Auf_BG-QM44";
       "UP_CM02.GP05".In.SRM_UV02_GP02_auf := "DB_PNOZ_IN_Out".In."SRM_Auf_BG-QM43" AND NOT "DB_PNOZ_IN_Out".In."SRM_Zu_BG-QM43";
       "UP_CM02.GP05".In.SRM_UV02_GP02_zu := "DB_PNOZ_IN_Out".In."SRM_Zu_BG-QM43" AND NOT "DB_PNOZ_IN_Out".In."SRM_Auf_BG-QM43";
       "UP_CM02.GP05".In."SRM_GP02.QM41_auf" := "E_SRM_GP02.QM41_auf" AND NOT "E_SRM_GP02.QM41_zu";
       "UP_CM02.GP05".In."SRM_GP01.QM14_auf" := "E_SRM_GP01.QM14_auf" AND NOT "E_SRM_GP01.QM14_zu";

       // Türen GP0x
       "UP_CM02.GP05".In.Tuer_zu_Seite_GP01 := "DB_PNOZ_IN_Out".In.Tuer_zu_Seite_GP01;
       "UP_CM02.GP05".In.Tuer_zu_vorn_GP01 := "DB_PNOZ_IN_Out".In.Tuer_zu_vorn_GP01;
       "UP_CM02.GP05".In.Tuer_zu_vorn_GP02 := "DB_PNOZ_IN_Out".In.Tuer_zu_vorn_GP02;

       // Leckagen Entsorgung
       "UP_CM02.GP05".In.Leckage_Doppelrohr_ok_BL26 := "E_LS_GP02.BL26";
       "UP_CM02.GP05".In.Leckage_Doppelschlauch_ok_BL33 := "E_LS_GP02.BL33";
       "UP_CM02.GP05".In.Leckage_Uml_Tunnel_ok_BL34 := "E_LS_GP01.BL34";
       "UP_CM02.GP05".In.Leckage_PFA_Uebergang_ok_BL16 := "E_LS_GP01.BL16";
       "UP_CM02.GP05".In.Leckage_PFA_Uebergang_ok_BL25 := "E_LS_GP02.BL25";

       "UP_CM02.GP05".In.Imp_Dfl := "E_Imp_GP02.BF02";
       "UP_CM02.GP05".In.Quitt_Al_Dfl := "DB_ANLAGE".IN.Quitt_Err;

       "UP_CM02.GP05".In.GW_p_UP := "E_GW_p_CM02.BP07";
       "UP_CM02.GP05".In.GW_p_UP := "E_GW_LF_CM02.BN04";
       "UP_CM02.GP05".In.GW_Dfl := "E_GW_Dfl_GP02.BF02";
       // TW senkt
       "UP_CM02.GP05".In.TW_senkt := ("DB_POS".POS[13].FW_Senkt OR "DB_POS".POS[14].FW_Senkt OR "DB_POS".POS[15].FW_Senkt
       OR "DB_POS".POS[16].FW_Senkt OR "DB_POS".POS[17].FW_Senkt OR "DB_POS".POS[18].FW_Senkt) AND "DI_FW_1".ZST.Mittig;

       // Frequenzumrichter [Index 5]
       "UP_CM02.GP05".In.FU_speed := "FU_In_Out".FU[5].PE.Speed;
       "UP_CM02.GP05".In.FU_betriebsbereit := "FU_In_Out".FU[5].PE.Statusbyte.Bereit;
       "UP_CM02.GP05".In.FU_Stoerung := "FU_In_Out".FU[5].PE.Statusbyte.Stoer;
       "UP_CM02.GP05".Param.SW_Hand := "Panel".UP_CM02.SW_Hand;
       "UP_CM02.GP05".Param.SW_Auto_AZ := "Panel".UP_CM02.SW_Auto_AZ;
       "UP_CM02.GP05".Param.SW_Auto_aAZ := "Panel".UP_CM02.SW_Auto_aAZ;

       // Hand
       "UP_CM02.GP05".In.Ein := "Panel".UP_CM02.Ein;
       // Auto
       "UP_CM02.GP05".In.Auto := "Panel".UP_CM02.Auto;
       // Betriebsart
       "UP_CM02.GP05".In.Betriebsart := "Panel".UP_CM02.BA;
       // Spülzeit
       "UP_CM02.GP05".Param.Spülzeit := DINT_TO_TIME(INT_TO_DINT("Panel".UP_CM02.Sp_Ventil.Sollzeit) * 1000);
       // Drucktest
       "UP_CM02.GP05".Param.DT_Druckaufbau := T#1m;
       "UP_CM02.GP05".Param.SW_Drucktest := "Panel".UP_CM02.Drucktest.Solldruck;
       "UP_CM02.GP05".Param.DT_Testzeit := DINT_TO_TIME(INT_TO_DINT("Panel".UP_CM02.Drucktest.Sollzeit) * 1000);

       //--> Panel
       "Panel".CM02.Niv_TGS := "UP_CM02.GP05".In.Niv_TLS;
       "Panel".CM02.Niv_Min := "UP_CM02.GP05".In.Niv_min;
       "Panel".CM02.Niv_max := "UP_CM02.GP05".In.Niv_max;
       "Panel".CM02.Niv_Uel := "UP_CM02.GP05".Mld.Niv_Ueberlauf;
       "Panel".CM02.GW_p_UP := "UP_CM02.GP05".Mld.GW_p_UP;
       "Panel".CM02.GW_LF_UP := "UP_CM02.GP05".Mld.GW_LF_UP;
       "Panel".CM02.Niv_Proz := "UP_CM02.GP05".Zst.Niveau;
       "Panel".UP_CM02.Sp_Ventil.Restzeit := TIME_TO_INT("UP_CM02.GP05".Zst.Restzeit_Spülen / 1000);
       "Panel".UP_CM02.Drucktest.Restzeit := TIME_TO_INT("UP_CM02.GP05".Zst.Restzeit_DT / 1000);
       "Panel".UP_CM02.Drucktest.Schritt := "UP_CM02.GP05".Zst.Status_DT;
       "Panel".UP_CM02.Status := "UP_CM02.GP05".Zst.Status_GP0x;
       "Panel".UP_CM02.speed := "UP_CM02.GP05".Zst.speed;
       "Panel".UP_CM02.Bedienung_Erlaubt := "UP_CM02.GP05".Zst.Bedienung_erlaubt;
   END_REGION
END_REGION

REGION Network 5 (SCL): CM03
   "UP_CM03.GP03".Param.Name := 'UP_CM03.GP03';
   // Niveaus
   "UP_CM03.GP03".In.Niv_TLS := "E_Niv_TLS_CM03.BL07";
   "UP_CM03.GP03".In.Niv_min := "E_Niv_Min_CM03.BL06";
   "UP_CM03.GP03".In.Frg_Niv_CM05 := NOT "Pu_CM05.GP11_DB".In."Niv_max_CM05.BL01" AND NOT "Pu_CM05.GP11_DB".In."Niv_Uel_CM05.BL05";
   "UP_CM03.GP03".In.ext_Freigabe := "E_Al_Gas_ok" AND NOT"E_Not-Strom";
   // Ist-Druck
   "UP_CM03.GP03".In.Druck_Pumpe := "Panel".IW."p_CM03.BP05";

   // Stellrückmeldungen
   "UP_CM03.GP03".In.SRM_Saugseite_auf := "E_SRM_CM03.QM33_auf" AND NOT "E_SRM_CM03.QM33_zu";
   "UP_CM03.GP03".In.SRM_Saugseite_zu := "E_SRM_CM03.QM33_zu" AND NOT "E_SRM_CM03.QM33_auf";
   "UP_CM03.GP03".In.SRM_Druckseite_auf := "E_SRM_CM03.QM34_auf" AND NOT "E_SRM_CM03.QM34_zu";
   "UP_CM03.GP03".In.SRM_Druckseite_zu := "E_SRM_CM03.QM34_zu" AND NOT "E_SRM_CM03.QM34_auf";

   "UP_CM03.GP03".In.GW_p_UP := "E_GW_p_CM03.BP05";
   // TW senkt
   "UP_CM03.GP03".In.TW_senkt := ("DB_POS".POS[7].FW_Senkt OR "DB_POS".POS[8].FW_Senkt OR "DB_POS".POS[9].FW_Senkt
   OR "DB_POS".POS[10].FW_Senkt OR "DB_POS".POS[11].FW_Senkt OR "DB_POS".POS[12].FW_Senkt) AND "DI_FW_1".ZST.Mittig;

   // Frequenzumrichter [Index 3]
   "UP_CM03.GP03".In.FU_speed := "FU_In_Out".FU[3].PE.Speed;
   "UP_CM03.GP03".In.FU_betriebsbereit := "FU_In_Out".FU[3].PE.Statusbyte.Bereit;
   "UP_CM03.GP03".In.FU_Stoerung := "FU_In_Out".FU[3].PE.Statusbyte.Stoer;
   "UP_CM03.GP03".Param.SW_Hand := "Panel".UP_CM03.SW_Hand;
   "UP_CM03.GP03".Param.SW_Auto_AZ := "Panel".UP_CM03.SW_Auto_AZ;
   "UP_CM03.GP03".Param.SW_Auto_aAZ := "Panel".UP_CM03.SW_Auto_aAZ;

   // Hand
   "UP_CM03.GP03".In.Ein := "Panel".UP_CM03.Ein;
   // Auto
   "UP_CM03.GP03".In.Auto := FALSE; // "Panel".UP_CM03.Auto;
   // Betriebsart
   "UP_CM03.GP03".In.Betriebsart := "Panel".UP_CM03.BA;
   // Spülzeit
   "UP_CM03.GP03".Param.Spülzeit := DINT_TO_TIME(INT_TO_DINT("Panel".UP_CM03.Sp_Ventil.Sollzeit) * 1000);
   // Drucktest
   "UP_CM03.GP03".Param.DT_Druckaufbau := T#1m;
   "UP_CM03.GP03".Param.SW_Drucktest := "Panel".UP_CM03.Drucktest.Solldruck;
   "UP_CM03.GP03".Param.DT_Testzeit := DINT_TO_TIME(INT_TO_DINT("Panel".UP_CM03.Drucktest.Sollzeit) * 1000);


   // --> Panel
   "Panel".CM03.Niv_TGS := "UP_CM03.GP03".In.Niv_TLS;
   "Panel".CM03.Niv_Min := "UP_CM03.GP03".In.Niv_min;
   "Panel".CM03.GW_p_UP := "UP_CM03.GP03".In.GW_p_UP;
   "Panel".CM03.Niv_Proz := "UP_CM03.GP03".Zst.Niveau;
   "Panel".UP_CM03.Sp_Ventil.Restzeit := TIME_TO_INT("UP_CM03.GP03".Zst.Restzeit_Spülen / 1000);
   "Panel".UP_CM03.Drucktest.Restzeit := TIME_TO_INT("UP_CM03.GP03".Zst.Restzeit_DT / 1000);
   "Panel".UP_CM03.Drucktest.Schritt := "UP_CM03.GP03".Zst.Status_DT;
   "Panel".UP_CM03.Status := "UP_CM03.GP03".Zst.Status_GP0x;
   "Panel".UP_CM03.speed := "UP_CM03.GP03".Zst.speed;
   "Panel".UP_CM03.Bedienung_Erlaubt := "UP_CM03.GP03".Zst.Bedienung_erlaubt;
END_REGION

REGION Network 6 (SCL): CM04
   "UP_CM04.GP06".Param.Name := 'UP_CM04.GP06';
   // Niveaus
   "UP_CM04.GP06".In.Niv_TLS := "E_Niv_TLS_CM04.BL14";
   "UP_CM04.GP06".In.Niv_min := "E_Niv_Min_CM04.BL13";
   "UP_CM04.GP06".In.Frg_Niv_CM05 := NOT "Pu_CM05.GP11_DB".In."Niv_max_CM05.BL01" AND NOT "Pu_CM05.GP11_DB".In."Niv_Uel_CM05.BL05";
   "UP_CM04.GP06".In.ext_Freigabe := "E_Al_Gas_ok" AND NOT "E_Not-Strom";
   // Ist-Druck
   "UP_CM04.GP06".In.Druck_Pumpe := "Panel".IW."p_CM04.BP08";

   // Stellrückmeldungen
   "UP_CM04.GP06".In.SRM_Saugseite_auf := "E_SRM_CM04.QM72_auf" AND NOT "E_SRM_CM04.QM72_zu";
   "UP_CM04.GP06".In.SRM_Saugseite_zu := "E_SRM_CM04.QM72_zu" AND NOT "E_SRM_CM04.QM72_auf";
   "UP_CM04.GP06".In.SRM_Druckseite_auf := "E_SRM_CM04.QM73_auf" AND NOT "E_SRM_CM04.QM73_zu";
   "UP_CM04.GP06".In.SRM_Druckseite_zu := "E_SRM_CM04.QM73_zu" AND NOT "E_SRM_CM04.QM73_auf";

   "UP_CM04.GP06".In.GW_p_UP := "E_GW_p_CM04.BP08";

   // TW senkt
   "UP_CM04.GP06".In.TW_senkt := ("DB_POS".POS[19].FW_Senkt OR "DB_POS".POS[20].FW_Senkt OR "DB_POS".POS[21].FW_Senkt
   OR "DB_POS".POS[22].FW_Senkt OR "DB_POS".POS[23].FW_Senkt OR "DB_POS".POS[24].FW_Senkt) AND "DI_FW_1".ZST.Mittig;

   // Frequenzumrichter [Index 6]
   "UP_CM04.GP06".In.FU_speed := "FU_In_Out".FU[6].PE.Speed;
   "UP_CM04.GP06".In.FU_betriebsbereit := "FU_In_Out".FU[6].PE.Statusbyte.Bereit;
   "UP_CM04.GP06".In.FU_Stoerung := "FU_In_Out".FU[6].PE.Statusbyte.Stoer;
   "UP_CM04.GP06".Param.SW_Hand := "Panel".UP_CM04.SW_Hand;
   "UP_CM04.GP06".Param.SW_Auto_AZ := "Panel".UP_CM04.SW_Auto_AZ;
   "UP_CM04.GP06".Param.SW_Auto_aAZ := "Panel".UP_CM04.SW_Auto_aAZ;

   // Hand
   "UP_CM04.GP06".In.Ein := "Panel".UP_CM04.Ein;
   // Auto
   "UP_CM04.GP06".In.Auto := FALSE; // "Panel".UP_CM04.Auto;
   // Betriebsart
   "UP_CM04.GP06".In.Betriebsart := "Panel".UP_CM04.BA;

   // Spülzeit
   "UP_CM04.GP06".Param.Spülzeit := DINT_TO_TIME(INT_TO_DINT("Panel".UP_CM04.Sp_Ventil.Sollzeit) * 1000);
   // Drucktest
   "UP_CM04.GP06".Param.DT_Druckaufbau := T#1m;
   "UP_CM04.GP06".Param.SW_Drucktest := "Panel".UP_CM04.Drucktest.Solldruck;
   "UP_CM04.GP06".Param.DT_Testzeit := DINT_TO_TIME(INT_TO_DINT("Panel".UP_CM04.Drucktest.Sollzeit) * 1000);

   // --> Panel
   "Panel".CM04.Niv_TGS := "UP_CM04.GP06".In.Niv_TLS;
   "Panel".CM04.Niv_Min := "UP_CM04.GP06".In.Niv_min;
   "Panel".CM04.GW_p_UP := "UP_CM04.GP06".In.GW_p_UP;
   "Panel".CM04.Niv_Proz := "UP_CM04.GP06".Zst.Niveau;
   "Panel".UP_CM04.Sp_Ventil.Restzeit := TIME_TO_INT("UP_CM04.GP06".Zst.Restzeit_Spülen / 1000);
   "Panel".UP_CM04.Drucktest.Restzeit := TIME_TO_INT("UP_CM04.GP06".Zst.Restzeit_DT / 1000);
   "Panel".UP_CM04.Drucktest.Schritt := "UP_CM04.GP06".Zst.Status_DT;
   "Panel".UP_CM04.Status := "UP_CM04.GP06".Zst.Status_GP0x;
   "Panel".UP_CM04.speed := "UP_CM04.GP06".Zst.speed;
   "Panel".UP_CM04.Bedienung_Erlaubt := "UP_CM04.GP06".Zst.Bedienung_erlaubt;
END_REGION

REGION Network 7 (SCL): CM05
   // Motorschutzschalter
   "Pu_CM05.GP11_DB".In.MSS_ok := "E_MSS_ok_CM05.GP11";
   // Druckschalter
   "Pu_CM05.GP11_DB".In.GW_p := "E_GW_p_CM05.BP09";
   // Ist-Druck
   "Pu_CM05.GP11_DB".In.Druck_Pumpe :="Panel".IW."p_CM05.BP09";

   // Niveaus
   "Pu_CM05.GP11_DB".In."Niv_max_CM05.BL01" := "E_Niv_max_CM05.BL01";
   "Pu_CM05.GP11_DB".In."Niv_min_CM05.BL02" := "E_Niv_min_CM05.BL02";
   "Pu_CM05.GP11_DB".In."Niv_TLS_CM05.BL03" := "E_Niv_TLS_CM05.BL03";
   "Pu_CM05.GP11_DB".In."Niv_Uel_CM05.BL05" :=  NOT "E_Niv_Uel_CM05.BL12";

   // Stellrückmeldungen
   "Pu_CM05.GP11_DB".In."SRM_CM05.QM61_auf" := "E_SRM_CM05.QM61_auf" AND NOT "E_SRM_CM05.QM61_zu";
   "Pu_CM05.GP11_DB".In."SRM_CM05.QM61_zu" := "E_SRM_CM05.QM61_zu" AND NOT "E_SRM_CM05.QM61_auf";
   "Pu_CM05.GP11_DB".In."SRM_CM05.QM64_auf" := "E_SRM_CM05.QM64_auf" AND NOT "E_SRM_CM05.QM64_zu";
   "Pu_CM05.GP11_DB".In."SRM_CM05.QM64_zu" := "E_SRM_CM05.QM64_zu"  AND NOT "E_SRM_CM05.QM64_auf";

   // Neutra
   "Pu_CM05.GP11_DB".In.AWA_ok := "E_AWA_ok";
   "Pu_CM05.GP11_DB".In.Frg_AWA := "E_Frg_AWA";
   // Hand
   "Pu_CM05.GP11_DB".In.Ein := "Panel".Pu_CM05.Ein;
   // Auto
   "Pu_CM05.GP11_DB".In.Auto := "Panel".Pu_CM05.Auto;
   // Betriebsart
   "Pu_CM05.GP11_DB".In.Betriebsart := "Panel".Pu_CM05.BA;
   // Spülzeit
   "Pu_CM05.GP11_DB".Param.Spülzeit := DINT_TO_TIME(INT_TO_DINT("Panel".Pu_CM05.Sp_Ventil.Sollzeit) * 1000);
   // Drucktest
   "Pu_CM05.GP11_DB".Param.DT_Druckaufbau := T#1m;
   "Pu_CM05.GP11_DB".Param.SW_Drucktest := "Panel".Pu_CM05.Drucktest.Solldruck;
   "Pu_CM05.GP11_DB".Param.DT_Testzeit := DINT_TO_TIME(INT_TO_DINT("Panel".Pu_CM05.Drucktest.Sollzeit) * 1000);

   // --> Panel
   "Panel".CM05.GW_p_Pu := "Pu_CM05.GP11_DB".In.GW_p;
   "Panel".CM05.Niv_Proz := "Pu_CM05.GP11_DB".Zst.Niveau;
   "Panel".CM05.Niv_TGS := "Pu_CM05.GP11_DB".In."Niv_TLS_CM05.BL03";
   "Panel".CM05.Niv_Min := "Pu_CM05.GP11_DB".In."Niv_min_CM05.BL02";
   "Panel".CM05.Niv_max := "Pu_CM05.GP11_DB".In."Niv_max_CM05.BL01";
   "Panel".CM05.Niv_Uel := "Pu_CM05.GP11_DB".In."Niv_Uel_CM05.BL05";
   "Panel".Pu_CM05.Sp_Ventil.Restzeit := TIME_TO_INT("Pu_CM05.GP11_DB".Zst.Restzeit_Spülen / 1000);
   "Panel".Pu_CM05.Drucktest.Restzeit := TIME_TO_INT("Pu_CM05.GP11_DB".Zst.Restzeit_DT / 1000);
   "Panel".Pu_CM05.Drucktest.Schritt := "Pu_CM05.GP11_DB".Zst.Status_DT;
   "Panel".Pu_CM05.Status := "Pu_CM05.GP11_DB".Zst.Status_GP11;
   "Panel".CM05.AWA_Bereit := "Pu_CM05.GP11_DB".In.AWA_ok;
   "Panel".CM05.Frg_Abpumpen := "Pu_CM05.GP11_DB".In.Frg_AWA;
   "Panel".Pu_CM05.Bedienung_Erlaubt := "Pu_CM05.GP11_DB".Zst.Bedienung_erlaubt;
END_REGION

REGION Network 8 (SCL): CL0x
   //CL01
   // Niveaus
   "Pu_CL01.GP08".In.Frg_Niv_CM05 :=  NOT "Pu_CM05.GP11_DB".In."Niv_max_CM05.BL01" AND NOT "Pu_CM05.GP11_DB".In."Niv_Uel_CM05.BL05";
   "Pu_CL01.GP08".In.Leckage_ok := "E_LS_CL01.BL28";
   // Hand
   "Pu_CL01.GP08".In.Ein :="Panel".Pu_CL01.Ein;
   // Auto
   "Pu_CL01.GP08".In.Auto := "Panel".Pu_CL01.Auto;
   // Betriebsart
   "Pu_CL01.GP08".In.Betriebsart := "Panel".Pu_CL01.BA;
   // Spülzeit
   "Pu_CL01.GP08".Param.Spülzeit := DINT_TO_TIME(INT_TO_DINT("Panel".Pu_CL01.Sp_Ventil.Sollzeit) * 1000);

   // --> Panel
   "Panel".CL0x."LS_CL01.BL28" := NOT "Pu_CL01.GP08".In.Leckage_ok;
   "Panel".CL0x.Niv_Proz_CL01 := "Pu_CL01.GP08".Zst.Niveau;
   "Panel".Pu_CL01.Sp_Ventil.Restzeit := TIME_TO_INT("Pu_CL01.GP08".Zst.Restzeit_Spülen / 1000);
   "Panel".Pu_CL01.Status := "Pu_CL01.GP08".Zst.Status_GP0x;
   "Panel".Pu_CL01.Bedienung_Erlaubt := "Pu_CL01.GP08".Zst.Bedienung_Erlaubt;

   //CL02
   // Niveaus
   "Pu_CL02.GP09".In.Frg_Niv_CM05 :=  NOT "Pu_CM05.GP11_DB".In."Niv_max_CM05.BL01" AND NOT "Pu_CM05.GP11_DB".In."Niv_Uel_CM05.BL05";
   "Pu_CL02.GP09".In.Leckage_ok := "E_LS_CL02.BL29";
   // Hand
   "Pu_CL02.GP09".In.Ein := "Panel".Pu_CL02.Ein;
   // Auto
   "Pu_CL02.GP09".In.Auto := "Panel".Pu_CL02.Auto;
   // Betriebsart
   "Pu_CL02.GP09".In.Betriebsart := "Panel".Pu_CL02.BA;
   // Spülzeit
   "Pu_CL02.GP09".Param.Spülzeit := DINT_TO_TIME(INT_TO_DINT("Panel".Pu_CL02.Sp_Ventil.Sollzeit) * 1000);

   // --> Panel
   "Panel".CL0x."LS_CL02.BL29" := NOT  "Pu_CL02.GP09".In.Leckage_ok;
   "Panel".CL0x.Niv_Proz_CL02 := "Pu_CL02.GP09".Zst.Niveau;
   "Panel".Pu_CL02.Sp_Ventil.Restzeit := TIME_TO_INT("Pu_CL02.GP09".Zst.Restzeit_Spülen / 1000);
   "Panel".Pu_CL02.Status := "Pu_CL02.GP09".Zst.Status_GP0x;
   "Panel".Pu_CL02.Bedienung_Erlaubt := "Pu_CL02.GP09".Zst.Bedienung_Erlaubt;
END_REGION

REGION Network 9 (SCL): GP01
   // Versorgung
   //Niveaus
   "Pu_GP01.GP13".In.Niv_min := "E_Niv_min_GP01.BL17";
   "Pu_GP01.GP13".In.Niv_max := NOT "E_Niv_max_GP01.BL20";
   "Pu_GP01.GP13".In.Niveau := INT_TO_USINT(REAL_TO_INT("Panel".IW."Niv_GP01.BL30"));
   // Leckagesensoren
   "Pu_GP01.GP13".In.Leckage_Pumpe_ok := NOT "E_LS_GP01.BL15";
   "Pu_GP01.GP13".In.Leckage_PFA_Uebergang_ok := "E_LS_GP01.BL16";
   "Pu_GP01.GP13".In.Leckage_Doppelrohr_ok := "E_LS_GP01.BL19";
   "Pu_GP01.GP13".In.Leckage_Uml_Tunnel_ok := "E_LS_GP01.BL34";
   "Pu_GP01.GP13".In.Leckage_Doppelschlauch_ok := TRUE; // nur GP02
   "Pu_GP01.GP13".In.kein_Gas_Alarm := "E_Al_Gas_ok";

   "Pu_GP01.GP13".In.Niv_Min_CM01 := "E_Niv_Min_CM01.BL03";
   "Pu_GP01.GP13".In.Niv_Max_CM01 := "E_Niv_Max_CM01.BL02";
   "Pu_GP01.GP13".In.Niv_Übervoll_CM01 := NOT "E_Niv_UeL_CM01.BL01";
   "Pu_GP01.GP13".In.Niv_Min_CM02 := "E_Niv_Min_CM02.BL10";
   "Pu_GP01.GP13".In.Niv_Max_CM02 := "E_Niv_Max_CM02.BL09";
   "Pu_GP01.GP13".In.Niv_Übervoll_CM02 := NOT "E_Niv_UeL_CM02.BL08";
   "Pu_GP01.GP13".In.Frg_Niv_CM05 := NOT "Pu_CM05.GP11_DB".In."Niv_max_CM05.BL01" AND NOT "Pu_CM05.GP11_DB".In."Niv_Uel_CM05.BL05";

   // Stellrückmeldungen
   "Pu_GP01.GP13".In.SRM_Saugseite_auf := "E_SRM_GP01.QM15_auf" AND NOT "E_SRM_GP01.QM15_zu";
   "Pu_GP01.GP13".In.SRM_Saugseite_zu := "E_SRM_GP01.QM15_zu" AND NOT "E_SRM_GP01.QM15_auf";
   "Pu_GP01.GP13".In.SRM_Druckseite_auf := "E_SRM_GP01.QM18_auf" AND NOT "E_SRM_GP01.QM18_zu";
   "Pu_GP01.GP13".In.SRM_Druckseite_zu := "E_SRM_GP01.QM18_zu" AND NOT "E_SRM_GP01.QM18_auf";
   "Pu_GP01.GP13".In.SRM_Eingang_Spülltg_auf := "E_SRM_GP01.QM16_auf" AND NOT "E_SRM_GP01.QM16_zu";
   "Pu_GP01.GP13".In.SRM_Eingang_Spülltg_zu := "E_SRM_GP01.QM16_zu" AND NOT "E_SRM_GP01.QM16_auf";
   "Pu_GP01.GP13".In.SRM_Ausgang_Spülltg_auf := "E_SRM_GP01.QM17_auf" AND NOT "E_SRM_GP01.QM17_zu";
   "Pu_GP01.GP13".In.SRM_Ausgang_Spülltg_zu := "E_SRM_GP01.QM17_zu" AND NOT "E_SRM_GP01.QM17_auf";
   "Pu_GP01.GP13".In.SRM_Versogung_UV01_auf := "E_SRM_GP01.QM22_auf" AND NOT "E_SRM_GP01.QM22_zu";
   "Pu_GP01.GP13".In.SRM_Versogung_UV01_zu := "E_SRM_GP01.QM22_zu" AND NOT "E_SRM_GP01.QM22_auf";
   "Pu_GP01.GP13".In.SRM_UV01_CM01_auf := "E_SRM_GP01.QM20_auf" AND NOT "E_SRM_GP01.QM20_zu";
   "Pu_GP01.GP13".In.SRM_UV01_CM01_zu := "E_SRM_GP01.QM20_zu" AND NOT "E_SRM_GP01.QM20_auf";
   "Pu_GP01.GP13".In.SRM_UV01_CM02_auf := "E_SRM_GP01.QM19_auf" AND NOT "E_SRM_GP01.QM19_zu";
   "Pu_GP01.GP13".In.SRM_UV01_CM02_zu := "E_SRM_GP01.QM19_zu" AND NOT "E_SRM_GP01.QM19_auf";

   "Pu_GP01.GP13".In.IBC_vorhanden := "E_S_IBC_GP01.BG21";
   "Pu_GP01.GP13".In.Tuer_vorn_zu := "DB_PNOZ_IN_Out".In.Tuer_zu_vorn_GP01;
   "Pu_GP01.GP13".In.Tuer_seitlich_zu := "DB_PNOZ_IN_Out".In.Tuer_zu_Seite_GP01;

   "Pu_GP01.GP13".In.GW_Dfl := "E_GW_Dfl_GP01.BF01";
   "Pu_GP01.GP13".In.Imp_Dfl := "E_Imp_GP01.BF01";
   "Pu_GP01.GP13".In.Quitt_Al_Dfl := "DB_ANLAGE".IN.Quitt_Err;
   "Pu_GP01.GP13".In.Dfl := "Panel".IW."Dfl_GP01.BF01";

   // Hand
   "Pu_GP01.GP13".In.Ein := "Panel".Pu_Vers_GP01.Ein;
   // Auto
   "Pu_GP01.GP13".In.Auto := "Panel".Pu_Vers_GP01.Auto;
   // Betriebsart
   "Pu_GP01.GP13".In.Betriebsart := "Panel".Pu_Vers_GP01.BA;
   // Spülzeit
   "Pu_GP01.GP13".Param.Spülzeit := DINT_TO_TIME(INT_TO_DINT("Panel".Pu_Vers_GP01.Sp_Ventil.Sollzeit) * 1000);

   // --> Panel
   "Panel".GP01.Niv_leer := "Pu_GP01.GP13".In.Niv_min;
   "Panel".GP01.Niv_max := "Pu_GP01.GP13".In.Niv_max;
   "Panel".GP01.IBC_vorhanden := "Pu_GP01.GP13".In.IBC_vorhanden;
   "Panel".GP01.Tür_zu_vorn := "Pu_GP01.GP13".In.Tuer_vorn_zu;
   "Panel".GP01.Tür_zu_seitlich := "Pu_GP01.GP13".In.Tuer_seitlich_zu;

   "Panel".GP01.LS_Pumpe := NOT "Pu_GP01.GP13".In.Leckage_Pumpe_ok;
   "Panel".GP01.LS_Doppelrohr_BL19 := NOT "Pu_GP01.GP13".In.Leckage_Doppelrohr_ok;
   "Panel".GP01.LS_PFA_Übergang := NOT "Pu_GP01.GP13".In.Leckage_PFA_Uebergang_ok;
   "Panel".GP01.LS_Uml_Tunnel := NOT "Pu_GP01.GP13".In.Leckage_Uml_Tunnel_ok;

   "Panel".GP01.Niv_Proz := "Pu_GP01.GP13".In.Niveau;

   "Panel".GP01.Versorgung := "Pu_GP01.GP13".In.Betriebsart < 4;
   "Panel".GP01.Entsorgung := "Pu_GP01.GP13".In.Betriebsart = 4;


   "Panel".Pu_Vers_GP01.Status := "Pu_GP01.GP13".Zst.Status_GP0x;
   "Panel".Pu_Vers_GP01.Sp_Ventil.Restzeit := TIME_TO_INT("Pu_GP01.GP13".Zst.Restzeit_Spülen / 1000);
   "Panel".Pu_Vers_GP01.Bedienung_Erlaubt := "Pu_GP01.GP13".Zst.Bedienung_erlaubt;
   //-----------------------------------------------------------------------------------------------------------------------------------------
   // Abpumpen
   // Niveaus
   "Pu_GP01.GP12".In.Frg_Niv_CM05 :=  NOT "Pu_CM05.GP11_DB".In."Niv_max_CM05.BL01" AND NOT "Pu_CM05.GP11_DB".In."Niv_Uel_CM05.BL05";
   "Pu_GP01.GP12".In.Leckage_ok := "E_LS_GP01.BL18";
   // Hand
   "Pu_GP01.GP12".In.Ein := "Panel".Pu_Entl_GP01.Ein;
   // Auto
   "Pu_GP01.GP12".In.Auto := "Panel".Pu_Entl_GP01.Auto;
   // Betriebsart
   "Pu_GP01.GP12".In.Betriebsart := "Panel".Pu_Entl_GP01.BA;
   // Spülzeit
   "Pu_GP01.GP12".Param.Spülzeit := DINT_TO_TIME(INT_TO_DINT("Panel".Pu_Entl_GP01.Sp_Ventil.Sollzeit) * 1000);

   // --> Panel
   "Panel".GP01.LS_PuSu := NOT "Pu_GP01.GP12".In.Leckage_ok;
   "Panel".Pu_Entl_GP01.Sp_Ventil.Restzeit := TIME_TO_INT("Pu_GP01.GP12".Zst.Restzeit_Spülen / 1000);
   "Panel".Pu_Entl_GP01.Status := "Pu_GP01.GP12".Zst.Status_GP0x;
   "Panel".Pu_Entl_GP01.Bedienung_Erlaubt := "Pu_GP01.GP12".Zst.Bedienung_Erlaubt;
END_REGION

REGION Network 10 (SCL): GP02
   // Versorgung
   //Niveaus
   "Pu_GP02.GP10".In.Niv_min := "E_Niv_min_GP02.BL24";
   "Pu_GP02.GP10".In.Niv_max := NOT "E_Niv_max_GP02.BL23";
   "Pu_GP02.GP10".In.Niveau := INT_TO_USINT(REAL_TO_INT("Panel".IW."Niv_GP02.BL31"));
   // Leckagesensoren
   "Pu_GP02.GP10".In.Leckage_Pumpe_ok := NOT "E_LS_GP02.BL27";
   "Pu_GP02.GP10".In.Leckage_PFA_Uebergang_ok := "E_LS_GP02.BL25";
   "Pu_GP02.GP10".In.Leckage_Doppelrohr_ok := "E_LS_GP01.BL19";
   "Pu_GP02.GP10".In.Leckage_Uml_Tunnel_ok := TRUE; // nur GP01
   "Pu_GP02.GP10".In.Leckage_Doppelschlauch_ok := "E_LS_GP02.BL32";
   "Pu_GP02.GP10".In.kein_Gas_Alarm := "E_Al_Gas_ok";

   "Pu_GP02.GP10".In.Niv_Min_CM01 := "E_Niv_Min_CM01.BL03";
   "Pu_GP02.GP10".In.Niv_Max_CM01 := "E_Niv_Max_CM01.BL02";
   "Pu_GP02.GP10".In.Niv_Übervoll_CM01 := NOT "E_Niv_UeL_CM01.BL01";
   "Pu_GP02.GP10".In.Niv_Min_CM02 := "E_Niv_Min_CM02.BL10";
   "Pu_GP02.GP10".In.Niv_Max_CM02 := "E_Niv_Max_CM02.BL09";
   "Pu_GP02.GP10".In.Niv_Übervoll_CM02 := NOT "E_Niv_UeL_CM02.BL08";
   "Pu_GP02.GP10".In.Frg_Niv_CM05 := NOT "Pu_CM05.GP11_DB".In."Niv_max_CM05.BL01" AND NOT "Pu_CM05.GP11_DB".In."Niv_Uel_CM05.BL05";

   // Stellrückmeldungen
   "Pu_GP02.GP10".In.SRM_Saugseite_auf := "E_SRM_GP02.QM38_auf" AND NOT "E_SRM_GP02.QM38_zu";
   "Pu_GP02.GP10".In.SRM_Saugseite_zu := "E_SRM_GP02.QM38_zu" AND NOT "E_SRM_GP02.QM38_auf";
   "Pu_GP02.GP10".In.SRM_Druckseite_auf := "E_SRM_GP02.QM40_auf" AND NOT "E_SRM_GP02.QM40_zu";
   "Pu_GP02.GP10".In.SRM_Druckseite_zu := "E_SRM_GP02.QM40_zu" AND NOT "E_SRM_GP02.QM40_auf";
   "Pu_GP02.GP10".In.SRM_Eingang_Spülltg_auf := "E_SRM_GP02.QM39_auf" AND NOT "E_SRM_GP02.QM39_zu";
   "Pu_GP02.GP10".In.SRM_Eingang_Spülltg_zu := "E_SRM_GP02.QM39_zu" AND NOT "E_SRM_GP02.QM39_auf";
   "Pu_GP02.GP10".In.SRM_Ausgang_Spülltg_auf := "E_SRM_GP02.QM42_auf" AND NOT "E_SRM_GP02.QM42_zu";
   "Pu_GP02.GP10".In.SRM_Ausgang_Spülltg_zu := "E_SRM_GP02.QM42_zu" AND NOT "E_SRM_GP02.QM42_auf";
   "Pu_GP02.GP10".In.SRM_Versogung_UV01_auf := "E_SRM_GP01.QM21_auf" AND NOT "E_SRM_GP01.QM21_zu";
   "Pu_GP02.GP10".In.SRM_Versogung_UV01_zu := "E_SRM_GP01.QM21_zu" AND NOT "E_SRM_GP01.QM21_auf";
   "Pu_GP02.GP10".In.SRM_UV01_CM01_auf := "E_SRM_GP01.QM20_auf" AND NOT "E_SRM_GP01.QM20_zu";
   "Pu_GP02.GP10".In.SRM_UV01_CM01_zu := "E_SRM_GP01.QM20_zu" AND NOT "E_SRM_GP01.QM20_auf";
   "Pu_GP02.GP10".In.SRM_UV01_CM02_auf := "E_SRM_GP01.QM19_auf" AND NOT "E_SRM_GP01.QM19_zu";
   "Pu_GP02.GP10".In.SRM_UV01_CM02_zu := "E_SRM_GP01.QM19_zu" AND NOT "E_SRM_GP01.QM19_auf";

   "Pu_GP02.GP10".In.IBC_vorhanden := "E_S_IBC_GP02.BG22";
   "Pu_GP02.GP10".In.Tuer_vorn_zu := "DB_PNOZ_IN_Out".In.Tuer_zu_vorn_GP02;
   "Pu_GP02.GP10".In.Tuer_seitlich_zu := TRUE;

   "Pu_GP02.GP10".In.GW_Dfl := "E_GW_Dfl_GP01.BF01";
   "Pu_GP02.GP10".In.Imp_Dfl := "E_Imp_GP01.BF01";
   "Pu_GP02.GP10".In.Quitt_Al_Dfl := "DB_ANLAGE".IN.Quitt_Err;
   "Pu_GP02.GP10".In.Dfl := "Panel".IW."Dfl_GP01.BF01";
   "Pu_GP02.GP10".In.Niveau := INT_TO_USINT(REAL_TO_INT("Panel".IW."Niv_GP02.BL31"));

   // Hand
   "Pu_GP02.GP10".In.Ein := "Panel".Pu_Vers_GP02.Ein;
   // Auto
   "Pu_GP02.GP10".In.Auto := "Panel".Pu_Vers_GP02.Auto;
   // Betriebsart
   "Pu_GP02.GP10".In.Betriebsart := "Panel".Pu_Vers_GP02.BA;
   // Spülzeit
   "Pu_GP02.GP10".Param.Spülzeit := DINT_TO_TIME(INT_TO_DINT("Panel".Pu_Vers_GP02.Sp_Ventil.Sollzeit) * 1000);

   // --> Panel
   "Panel".GP02.Niv_leer := "Pu_GP02.GP10".In.Niv_min;
   "Panel".GP02.Niv_max := "Pu_GP02.GP10".In.Niv_max;
   "Panel".GP02.IBC_vorhanden := "Pu_GP02.GP10".In.IBC_vorhanden;

   "Panel".GP02.Tür_zu_seitlich := "Pu_GP02.GP10".In.Tuer_seitlich_zu;

   "Panel".GP02.LS_Doppelschlauch_BL32 := NOT "E_LS_GP02.BL32";
   "Panel".GP02.LS_Doppelschlauch_BL33 := NOT "E_LS_GP02.BL33";
   "Panel".GP02.LS_Doppelrohr_BL26 := NOT "E_LS_GP02.BL26";
   "Panel".GP02.LS_Pumpe := NOT "Pu_GP02.GP10".In.Leckage_Pumpe_ok;
   "Panel".GP02.LS_PFA_Übergang := NOT "Pu_GP02.GP10".In.Leckage_PFA_Uebergang_ok;
   "Panel".GP02.Niv_Proz := "Pu_GP02.GP10".In.Niveau;

   "Panel".GP02.Versorgung := "Pu_GP02.GP10".In.Betriebsart < 4;
   "Panel".GP02.Entsorgung := "Pu_GP02.GP10".In.Betriebsart = 4;

   "Panel".Pu_Vers_GP02.Status := "Pu_GP02.GP10".Zst.Status_GP0x;
   "Panel".Pu_Vers_GP02.Sp_Ventil.Restzeit := TIME_TO_INT("Pu_GP02.GP10".Zst.Restzeit_Spülen / 1000);
   "Panel".Pu_Vers_GP02.Bedienung_Erlaubt := "Pu_GP02.GP10".Zst.Bedienung_erlaubt;
   //-----------------------------------------------------------------------------------------------------------------------------------------

   // Abpumpen
   // Niveaus
   "Pu_GP02.GP07".In.Frg_Niv_CM05 :=  NOT "Pu_CM05.GP11_DB".In."Niv_max_CM05.BL01" AND NOT "Pu_CM05.GP11_DB".In."Niv_Uel_CM05.BL05";
   "Pu_GP02.GP07".In.Leckage_ok := "E_LS_GP02.BL21";
   // Hand
   "Pu_GP02.GP07".In.Ein := "Panel".Pu_Entl_GP02.Ein;
   // Auto
   "Pu_GP02.GP07".In.Auto := "Panel".Pu_Entl_GP02.Auto;
   // Betriebsart
   "Pu_GP02.GP07".In.Betriebsart := "Panel".Pu_Entl_GP02.BA;
   // Spülzeit
   "Pu_GP02.GP07".Param.Spülzeit := DINT_TO_TIME(INT_TO_DINT("Panel".Pu_Entl_GP02.Sp_Ventil.Sollzeit) * 1000);

   // --> Panel
   "Panel".GP02.LS_PuSu := NOT "Pu_GP02.GP07".In.Leckage_ok;
   "Panel".Pu_Entl_GP02.Sp_Ventil.Restzeit := TIME_TO_INT("Pu_GP02.GP07".Zst.Restzeit_Spülen / 1000);
   "Panel".Pu_Entl_GP02.Status := "Pu_GP02.GP07".Zst.Status_GP0x;
   "Panel".Pu_Entl_GP02.Bedienung_Erlaubt := "Pu_GP02.GP07".Zst.Bedienung_Erlaubt;
END_REGION
END_FUNCTION
